{attribute 'qualified_only'}
VAR_GLOBAL
	// udiDI%65.0_A4_5
	{attribute 'OPC.UA.DA' := '1'} // für OPC UA freigeben
	VSG_Enc_vertikal_I1 AT %I*: UDINT;
	{attribute 'OPC.UA.DA' := '1'} // für OPC UA freigeben
	// udiDI%71.0_A4_5
	VSG_Enc_vertikal_I2 AT %I*: UDINT;
	{attribute 'OPC.UA.DA' := '1'} // für OPC UA freigeben
	// udiDI%77.0_A4_5
	VSG_Enc_horizontal_I1 AT %I*: UDINT;
	{attribute 'OPC.UA.DA' := '1'} // für OPC UA freigeben
	// udiDI%83.0_A4_5
	VSG_Enc_horizontal_I2 AT %I*: UDINT;
	{attribute 'OPC.UA.DA' := '1'} // für OPC UA freigeben
	// udiDI%89.0_A4_5
	VSG_Enc_drehen_I1 AT %I*: UDINT;
	{attribute 'OPC.UA.DA' := '1'} // für OPC UA freigeben
	// udiDI%95.0_A4_5
	VSG_Enc_drehen_I2 AT %I*: UDINT;
	{attribute 'OPC.UA.DA' := '1'} // für OPC UA freigeben
	// xDI%138.1_A4_2
	VSG_Ref_Schalter_vertikal AT %I*: BOOL;
	{attribute 'OPC.UA.DA' := '1'} // für OPC UA freigeben
	// xDI%138.2_A4_2
	VSG_Ref_Schalter_horizontal AT %I*: BOOL;
	{attribute 'OPC.UA.DA' := '1'} // für OPC UA freigeben
	// xDI%138.3_A4_2
	VSG_Ref_Schalter_drehen AT %I*: BOOL;
	{attribute 'OPC.UA.DA' := '1'} // für OPC UA freigeben
	// xDO%113.6_A4_4
	VSG_MOT_vertikal_hoch AT %Q*: BOOL;
	{attribute 'OPC.UA.DA' := '1'} // für OPC UA freigeben
	// xDO%113.7_A4_4
	VSG_MOT_vertikal_runter AT %Q*: BOOL;
	{attribute 'OPC.UA.DA' := '1'} // für OPC UA freigeben
	// xDO%114.0_A4_4
	VSG_MOT_horizontal_rueckwaerts AT %Q*: BOOL;
	{attribute 'OPC.UA.DA' := '1'} // für OPC UA freigeben
	// xDO%114.1_A4_4
	VSG_MOT_horizontal_vorwaerts AT %Q*: BOOL;
	{attribute 'OPC.UA.DA' := '1'} // für OPC UA freigeben
	// xDO%114.2_A4_4
	VSG_MOT_drehen_CW AT %Q*: BOOL;
	{attribute 'OPC.UA.DA' := '1'} // für OPC UA freigeben
	// xDO%114.3_A4_4
	VSG_MOT_drehen_CCW AT %Q*: BOOL;
	{attribute 'OPC.UA.DA' := '1'} // für OPC UA freigeben
	// xDO%114.4_A4_8
	VSG_Kompressor AT %Q*: BOOL;
	{attribute 'OPC.UA.DA' := '1'} // für OPC UA freigeben
	// xDO%114.5_A4_5
	{attribute 'OPC.UA.DA' := '1'} // für OPC UA freigeben
	VSG_MV_Vakuum AT %Q*: BOOL;
	{attribute 'OPC.UA.DA' := '1'} // für OPC UA freigeben
	VSG_K1_4_Zaehler_Zuruecksetzen AT %Q*: BOOL;
	{attribute 'OPC.UA.DA' := '1'} // für OPC UA freigeben
	VSG_K1_5_Zaehler_Zuruecksetzen AT %Q*: BOOL;
	{attribute 'OPC.UA.DA' := '1'} // für OPC UA freigeben
	VSG_K1_3_Zaehler_Zuruecksetzen AT %Q*: BOOL;
END_VAR

(* stored: Version 1.1.0.1, ProductVersion 3.1.4026.18
   GVL GVL_VSG: Id {e0027df7-4efe-4e0c-b7b0-8eacf699165e} *)
